{attribute 'GeneratedUsingTerminal: EP6090-0000-0017'}
{attribute addProperty BoxType "EP6090-0000-0017"}
{attribute addProperty Id "StatusAT %I*Status_E3E7FD126"}
{attribute addProperty CRC "3773007075"}
{attribute addProperty Size "6"}
TYPE DIS_Inputs_E0E384E3 EXTENDS InputBase_8311D824 :
STRUCT
	{attribute addProperty Name "Status"}
	Status AT %I* : Status_E3E7FD12;
END_STRUCT
END_TYPE

(* stored: Version 1.2.0.0, ProductVersion 3.1.4024.11
   DUT DIS_Inputs_E0E384E3: Id {cb37b1b4-5679-423c-8f75-f05892639a2a} *)
